ABB RAPID module: Module1.mod

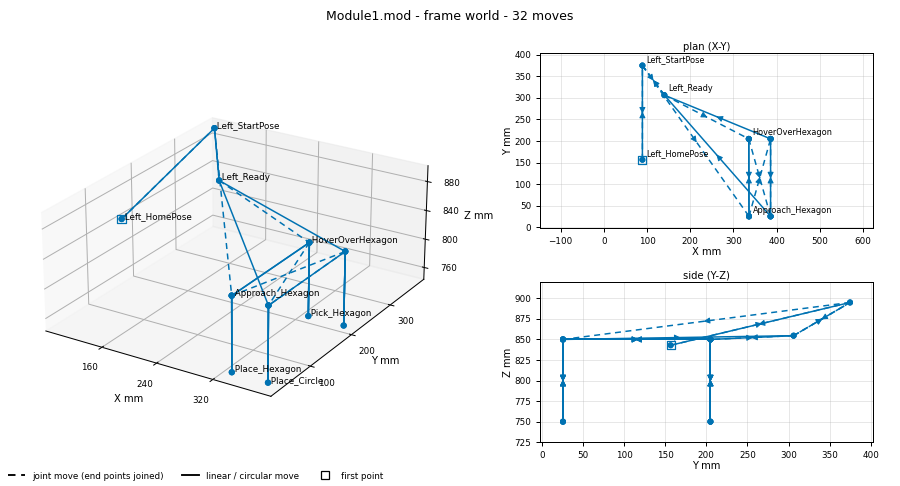
[picture p0: tool path of Module1.mod in frame world, 32 of 32 moves have a stored position in this frame; points joined in program order, loops and branches not executed]
MODULE Module1
    CONST robtarget Left_HomePose:=[[89.387946423,156.622117957,842.913470217],[0.066010726,0.842420918,-0.111214912,0.523068661],[0,0,0,4],[101.964427132,9E+09,9E+09,9E+09,9E+09,9E+09]];
    CONST robtarget Left_StartPose:=[[89.389099881,374.790605689,894.969255092],[0.004761475,0.997945931,-0.011658513,-0.062811825],[0,1,-2,4],[101.861696088,9E+09,9E+09,9E+09,9E+09,9E+09]];
    CONST robtarget Left_Ready:=[[140.285116063,306.177691778,854.594529304],[-0.000000074,1,-0.000000247,-0.000000145],[0,-2,-2,4],[137.310759068,9E+09,9E+09,9E+09,9E+09,9E+09]];
    CONST robtarget HoverOverHexagon:=[[0,0,100],[0,1,0,0],[0,-2,-2,4],[101.964427132,9E+09,9E+09,9E+09,9E+09,9E+09]];
    CONST robtarget Pick_Hexagon:=[[0,0,0],[0,1,0,0],[-1,-2,-2,4],[101.964427132,9E+09,9E+09,9E+09,9E+09,9E+09]];
    CONST robtarget Approach_Hexagon:=[[-25.29,25.649,130],[0,1,0,0],[-1,-2,-2,4],[101.964427132,9E+09,9E+09,9E+09,9E+09,9E+09]];
    CONST robtarget Place_Hexagon:=[[-25.29,25.649,30],[0,1,0,0],[-1,-2,-2,4],[101.964427132,9E+09,9E+09,9E+09,9E+09,9E+09]];
    CONST robtarget HoverOverCircle:=[[-0.001,-0.002,100],[0,1,0,0],[-1,2,2,4],[101.964427132,9E+09,9E+09,9E+09,9E+09,9E+09]];
    CONST robtarget Pick_Circle:=[[-0.001,-0.002,0],[0,1,0,0],[0,0,0,0],[101.964427132,9E+09,9E+09,9E+09,9E+09,9E+09]];
    CONST robtarget Approach_Circle:=[[24.71,25.649,130],[0,1,0,0],[0,0,0,0],[101.964427132,9E+09,9E+09,9E+09,9E+09,9E+09]];
    CONST robtarget Place_Circle:=[[24.71,25.649,30],[0,1,0,0],[0,0,0,0],[101.964427132,9E+09,9E+09,9E+09,9E+09,9E+09]];
    PROC Path_10()
        ConfJ\Off;
        ConfL\Off;
        MoveJ Left_HomePose,v100,fine,Servo\WObj:=LeftArm;
        MoveJ Left_StartPose,v100,fine,Servo\WObj:=LeftArm;
        MoveJ Left_Ready,v100,fine,Servo\WObj:=LeftArm;
        MoveJ HoverOverHexagon,v100,fine,Servo\WObj:=HexagonObj;
        MoveL Pick_Hexagon,v100,fine,Servo\WObj:=HexagonObj;
        g_GripIn;
        WaitTime 1;
        MoveL HoverOverHexagon,v100,fine,Servo\WObj:=HexagonObj;
        MoveL Approach_Hexagon,v100,fine,Servo\WObj:=LeftMainHolder;
        MoveL Place_Hexagon,v100,fine,Servo\WObj:=LeftMainHolder;
        g_GripOut;
        WaitTime 1;
        MoveL Approach_Hexagon,v100,fine,Servo\WObj:=LeftMainHolder;
        MoveJ HoverOverCircle,v100,fine,Servo\WObj:=CircleObj;
        MoveL Pick_Circle,v100,fine,Servo\WObj:=CircleObj;
        g_GripIn;
        WaitTime 1;
        MoveL HoverOverCircle,v100,fine,Servo\WObj:=CircleObj;
        MoveJ Approach_Circle,v100,fine,Servo\WObj:=LeftMainHolder;
        MoveL Place_Circle,v100,fine,Servo\WObj:=LeftMainHolder;
        g_GripOut;
        WaitTime 1;
        MoveL Approach_Circle,v100,fine,Servo\WObj:=LeftMainHolder;
        MoveL Left_Ready,v100,fine,Servo\WObj:=LeftArm;
        MoveJ Left_StartPose,v100,fine,Servo\WObj:=LeftArm;
        MoveJ Approach_Hexagon,v100,fine,Servo\WObj:=LeftMainHolder;
        MoveL Place_Hexagon,v100,fine,Servo\WObj:=LeftMainHolder;
        g_GripIn;
        WaitTime 1;
        MoveL Approach_Hexagon,v100,fine,Servo\WObj:=LeftMainHolder;
        MoveL HoverOverHexagon,v100,fine,Servo\WObj:=HexagonObj;
        MoveL Pick_Hexagon,v100,fine,Servo\WObj:=HexagonObj;
        g_GripOut;
        WaitTime 1;
        MoveL HoverOverHexagon,v100,fine,Servo\WObj:=HexagonObj;
        MoveJ Approach_Circle,v100,fine,Servo\WObj:=LeftMainHolder;
        MoveL Place_Circle,v100,fine,Servo\WObj:=LeftMainHolder;
        g_GripIn;
        WaitTime 1;
        MoveL Approach_Circle,v100,fine,Servo\WObj:=LeftMainHolder;
        MoveL HoverOverCircle,v100,fine,Servo\WObj:=CircleObj;
        MoveL Pick_Circle,v100,fine,Servo\WObj:=CircleObj;
        g_GripOut;
        WaitTime 1;
        MoveL HoverOverCircle,v100,fine,Servo\WObj:=CircleObj;
        MoveL Left_Ready,v100,fine,Servo\WObj:=LeftArm;
        MoveJ Left_StartPose,v100,fine,Servo\WObj:=LeftArm;
        MoveL Left_HomePose,v100,fine,Servo\WObj:=LeftArm;
    ENDPROC
ENDMODULE
